INTERFACE ITF_MCMachineControl EXTENDS ITF_BaseTopElement

END_INTERFACE

(* stored: Version 1.1.0.1
   Itf ITF_MCMachineControl: Id {3df9f3b2-e7e8-0a37-055d-5ffd5d1b0cac} *)
